FUNCTION_BLOCK paloma
VAR_INPUT
	

END_VAR
VAR_OUTPUT
END_VAR
VAR

	VarAve: Ave;
END_VAR

END_FUNCTION_BLOCK

(* stored: Version 1.1.0.1, ProductVersion 3.1.4024.12
   POU paloma: Id {4ee7cdcc-a5a0-41b5-8c16-6399fbd38581}, SpecialFunc None *)
